Staubli VAL3: _sendJoint.pgx

program _sendJoint()
begin
  jCurrent = herej()

  sioSet(siTcpIpJoint, jCurrent.j1)
  sioSet(siTcpIpJoint, jCurrent.j2)
  sioSet(siTcpIpJoint, jCurrent.j3)
  sioSet(siTcpIpJoint, jCurrent.j4)
  sioSet(siTcpIpJoint, jCurrent.j5)
  sioSet(siTcpIpJoint, jCurrent.j6)
end
